TYPE stBH0JPL_Line EXTENDS stPIM_LineEventsModule :
STRUCT

	{attribute 'OPC.UA.DA' := '1'}
	stStation_BH0JPL01 : stPIM_StationEventsModule_3_Machine;
END_STRUCT
END_TYPE

(* stored: Version 1.1.0.1, ProductVersion 3.1.4024.15
   DUT stBH0JPL_Line: Id {ff09e214-b852-4fe2-acf6-6c547739883e} *)
